TYPE (* Setpoint Parameters for Variable Air Volume Controller *)
  (* Standard: 61499-1; ApplicationDomain: HVAC *)
  (* Version 0.2, 2006-05-12, JHC, Holobloc Inc, Corrected UnoccHtgSP from BOOL to REAL. *)
  (* Version 0.1, 2006-05-07, JHC, Holobloc Inc, Updated tag number to avoid conflict with COLOR. *)
  (* Version 0.0, 2006-04-04, JHC, Holobloc Inc *)
  (* Compiler header: package fb.rt.hvac; *)
  (* Compiler Java Sun JDK 1.5.0 *)
  (* ASN.1 tag PRIVATE 3 *)
  VAV_SP : STRUCT
    SP : REAL; (* Cooling setpoint. May be modified by the Temperature Setpoint (AI) as an offset *)
    UnoccSP : REAL; (* Unoccupied cooling setpoint.  The offset between SP and UnoccSP will remain the same *)
    StandbySP : REAL; (* Standby cooling setpoint. The offset between SP and StandbySP will remain the same *)
    HeatingSP : REAL; (* Occupied heating setpoint.  The offset between SP and HeatingSP will remain the same *)
    StandbyHtgSP : REAL; (* Standby heating setpoint. The offset between SP and StandbySP will remain the same *)
    UnoccHtgSP : REAL; (* Unoccupied heating setpoint. The offset between SP and UnoccHtgSP will remain the same *)
  END_STRUCT;
END_TYPE
